// TIA Portal V18 export
DATA_BLOCK "ALARM_DB"   // DB6
VERSION : 0.1
// stored: AutoNumber true, DBAccessibleFromOPCUA true, InstanceOfName ALARM, InstanceOfType FB
"ALARM"
   // VAR
   //    P1 : Bool;
   //    P2 : Bool;
   //    P3 : Bool;
   //    P4 : Bool;
   //    P5 : Bool;
   //    P6 : Bool;
   //    P7 : Bool;
   //    P8 : Bool;
   //    P9 : Bool;
   //    P10 : Bool;
   //    P11 : Bool;
   //    P12 : Bool;
   //    P13 : Bool;
   //    P14 : Bool;
   //    P15 : Bool;
   //    P16 : Bool;
   //    P17 : Bool;
   //    P18 : Bool;
   //    P19 : Bool;
   // END_VAR
BEGIN
END_DATA_BLOCK
